// TIA Portal V17 export
// export: Created 2026-04-13T11:12:43.2212045Z, ExportSetting WithDefaults, DisplayName Totally Integrated Automation Portal, DisplayVersion V17 Update 4, DisplayName TIA Portal Openness, DisplayVersion V17 Update 4, DisplayName TIA Portal Version Control Interface, DisplayVersion V17, DisplayName SINAMICS Startdrive Advanced, DisplayVersion V17, DisplayName SINAMICS Startdrive G130, G150, S120, S150, SINAMICS MV, S210, DisplayVersion V17, DisplayName SINAMICS Startdrive G110M, G120, G120C, G120D, G120P, G115D, DisplayVersion V17, DisplayName STEP 7 Professional, DisplayVersion V17 Update 4, DisplayName STEP 7 Safety, DisplayVersion V17, DisplayName WinCC Professional, DisplayVersion V17 Update 4
FUNCTION_BLOCK "0-模拟量输入2PID"   // FB79, SCL
{ S7_Optimized_Access := 'TRUE' }
VERSION : 0.1
// stored: AutoNumber true, IsIECCheckEnabled false, IsRetainMemResEnabled false, MemoryReserve 100, SetENOAutomatically false, UDAEnableTagReadback false
   VAR_INPUT
      AM : Bool := TRUE;   // 手动调节: 0,手动; 1,自动.
      ManualValue : Real;   // 手动调节输出值:0-100%.
      Enable : Bool;   // 自动调节使能. 1,启用; 0,不启用.
      Mode : Int := 1;   // 控制模式: 0,制热;1,制冷; 2,输出0.
      Setpoint : Real;   // 控制目标值
      Input : Real;   // 控制实际值
      ControlledObject_FB : Real;   // 受控对象实际值反馈(开度/频率...)
      Kp : Real;   // 比例系数(大于零实数)
      DeadZone : Real;   // 死区
      MAX : Real := 100.0;   // 上限
      MIN : Real;   // 下限
   END_VAR
   VAR_OUTPUT
      Output : Real;   // 受控对象输出值
   END_VAR
   VAR
      AutoValue : Real;
      output_Temp { ExternalAccessible := 'False'; ExternalVisible := 'False'; ExternalWritable := 'False'} : Real;
      RT_C : DInt;
   END_VAR
BEGIN
   IF  #AM AND #Enable THEN
       IF (#Mode=1) AND (ABS(#Input - #Setpoint) > #DeadZone) THEN
           #AutoValue := #ControlledObject_FB + #Kp * (#Input - #Setpoint) / 100;
       ELSIF (#Mode=0) AND (ABS(#Input - #Setpoint) > #DeadZone) THEN
           #AutoValue := #ControlledObject_FB - #Kp * (#Input - #Setpoint) / 100;
       ELSIF (#Mode=2) THEN
           #AutoValue := 0;
       ELSE
           #AutoValue := #ControlledObject_FB;
       END_IF;
   END_IF;

   IF NOT #AM THEN
       #output_Temp := #ManualValue;
   ELSE
       #output_Temp := #AutoValue;
   END_IF;

   IF #output_Temp >= #MAX THEN
       #Output := #MAX;
   ELSIF #output_Temp <= #MIN THEN
       #Output := #MIN;
   ELSE
       #Output := #output_Temp;
   END_IF;
END_FUNCTION_BLOCK
